INTERFACE I_LIGHT

METHOD Off
VAR_INPUT
END_VAR
END_METHOD

METHOD On
VAR_INPUT
END_VAR
END_METHOD

END_INTERFACE

(* stored: Version 1.1.0.1, ProductVersion 3.1.4024.12
   Itf I_LIGHT: Id {4d9d1918-5b33-47ec-8716-3a268df7d304}
   Method Off: Id {a800c40d-1265-499e-be2e-d11b1168d657}
   Method On: Id {a351c6d1-99ba-4366-bc04-9cafc55968ec} *)
